PROGRAM Speicher_leeren
VAR
	m:INT;
END_VAR

IF xPunkt_geaendert = TRUE OR (ILC_EinAus = FALSE AND MasterStart = TRUE) THEN
	FOR m := 0 TO 2000 BY 1 DO
		u_Old[m]:= 0;
		e_Old[m]:= 0;
		count := 0;
	END_FOR
	LernenFertig := FALSE;
	ILC_Out := 0;
	alt_xPunkt := xPunkt;
END_IF

END_PROGRAM

(* stored: Version 1.1.0.1, ProductVersion 3.1.4024.11
   POU Speicher_leeren: Id {b6bb0a27-ac79-466e-9144-05df1bef55f8}, SpecialFunc None *)
